FUNCTION CheckDivLReal  : LREAL
VAR_INPUT
	divisor : LREAL;
END_VAR
VAR
END_VAR

IF divisor = 0 THEN
        CheckDivReal := 1E-10;
ELSE
        CheckDivReal := divisor;
END_IF

END_FUNCTION

(* stored: Version 1.1.0.1, ProductVersion 3.1.4022.18
   POU CheckDivLReal: Id {28014d14-ae8d-48a8-8a5c-a8c352b954ff}, SpecialFunc None *)
